{ attribute 'allowImplicitAccess'}
TYPE ST_System_Control :
STRUCT
	control				: ST_ControlVars;
	Operation			: ST_OperationVars;
	SoftSettings		: ST_SoftSettings;
	HardSettings		: ST_Hardsettings;
END_STRUCT
END_TYPE

(* stored: Version 1.1.0.1, ProductVersion 3.1.4026.18
   DUT ST_System_Control: Id {c5705078-6fd9-44e7-a554-80ecc7a93178} *)
